Staubli VAL3: TrianglePoint.pgx

public program TrianglePoint(trsf& x_trSource[], trsf& x_trDest[], bool& x_bRes)
  local frame l_fFrame
  local trsf l_trCenter
  local num l_nDia
  local point l_p
  local trsf l_trBuff[3]
begin
  //三角形三点
  call Inscribedcircle(x_trSource,l_trCenter,l_nDia,x_bRes)
  if !x_bRes
    return
  endIf
      //圆心点
  x_trDest[20]=l_trCenter

  call SetFrame(x_trSource,l_fFrame,x_bRes)
  if !x_bRes
    return
  endIf

  l_p.trsf=l_trCenter
  link(l_p,world)
  l_p.trsf=position(l_p,l_fFrame)
  l_p.trsf.y=0
  link(l_p,l_fFrame)
  x_trDest[0]=position(l_p,world)

  x_trDest[1]=x_trSource[1]
  x_trDest[2]=x_trSource[2]
  x_trDest[3]=x_trSource[0]
  x_trDest[4]=x_trDest[0]

  for l_nDia=0 to 4
    x_trDest[l_nDia].rx= x_trDest[0].rx
    x_trDest[l_nDia].ry = x_trDest[0].ry
    x_trDest[l_nDia].rz= x_trDest[0].rz
  endFor



end
